FUNCTION_BLOCK CIRCULAR_VELOCITY (* Circular velocity equations *)
  (* Standard: 61499-2 *)
  (* Version 1.0, 02-05-12, GASR, Universidade do Estado de Santa Catarina *)
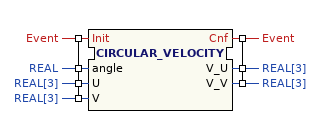
  EVENT_INPUT
    Init WITH angle, U, V;
  END_EVENT
  EVENT_OUTPUT
    Cnf WITH V_U, V_V;
  END_EVENT
  VAR_INPUT
    angle : REAL;
    U : ARRAY [0..2] OF REAL;
    V : ARRAY [0..2] OF REAL;
  END_VAR
  VAR_OUTPUT
    V_U : ARRAY [0..2] OF REAL;
    V_V : ARRAY [0..2] OF REAL;
  END_VAR
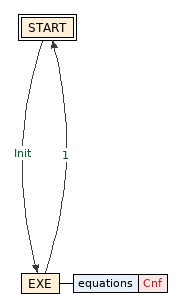
  EC_STATES
    START;
    EXE : equations -> Cnf;
  END_STATES
  EC_TRANSITIONS
    START TO EXE := Init;
    EXE TO START := 1;
  END_TRANSITIONS
  ALGORITHM equations IN Lua:
V_U[1] = U[1]*angle
V_U[2] = U[2]*angle
V_U[3] = U[3]*angle
V_V[1] = V[1]*angle
V_V[2] = V[2]*angle
V_V[3] = V[3]*angle
  END_ALGORITHM
END_FUNCTION_BLOCK
